{attribute addProperty BoxType "EL2878-0005-0016"}
{attribute addProperty Id "DiagnosticAT %I*Diagnostic_4CD4E3A2810ChannelAT %Q*ARRAY[0..7] OF Channel_7F374EB06480WcStateAT %I*WcState_98A4DF7520.250InfoDataAT %I*InfoData_192954DE1620"}
{attribute addProperty CRC "570157600"}
{attribute addProperty SizeInBites "90"}
{attribute addProperty SizeInBytes "11.25"}
TYPE EL2878_3D5C112B :
STRUCT
	{attribute addProperty Name "Diagnostic"}
	Diagnostic : Diagnostic_4CD4E3A2;
	{attribute addProperty Name "Channel"}
	Channel : ARRAY[0..7] OF Channel_7F374EB0;
	{attribute addProperty Name "WcState"}
	WcState : WcState_98A4DF75;
	{attribute addProperty Name "InfoData"}
	InfoData : InfoData_192954DE;
END_STRUCT
END_TYPE

(* stored: Version 1.2.0.0, ProductVersion 3.1.4024.9
   DUT EL2878_3D5C112B: Id {e649338b-4cba-4952-92ec-8969cf513f40} *)
